{attribute 'GeneratedUsingTerminal: EL6001--0000'}
{attribute addProperty BoxType "EL6001--0000"}
{attribute addProperty Id "StatusAT %I*UINT2Data_InAT %I*ARRAY[0..21] OF USINT22"}
{attribute addProperty CRC "1367962124"}
{attribute addProperty Size "24"}
TYPE Inputs_6C2FC202 :
STRUCT
	{attribute addProperty Name "Status"}
	Status AT %I* : UINT;
	{attribute addProperty Name "Data_In"}
	Data_In AT %I* : ARRAY[0..21] OF USINT;
END_STRUCT
END_TYPE

(* stored: Version 1.2.0.0, ProductVersion 3.1.4024.9
   DUT Inputs_6C2FC202: Id {7d653af9-a1e2-4020-8ef9-bcd3de4d5f92} *)
